// TIA Portal V20 export
DATA_BLOCK "DB_OPC_Laser"   // DB125
{ S7_Optimized_Access := 'TRUE' }
// stored: MemoryReserve 100
   VAR
      Scanner : Struct
         In : Struct
            CheckNumber : Byte;
            Ready : Bool;
            Status : DInt;
            StatusDescription : String;
         END_STRUCT;
         Out : Struct
            Parameters : Struct
               IsFirstJobOfPiece : Bool;
               StationNumber : Byte;
               HoleNumber : DInt;
               JobListName : String;
               JobName : String;
               MeasureZ : LReal;
            END_STRUCT;
            RequestJob : Bool;
            CheckNumber : Byte;
         END_STRUCT;
      END_STRUCT;
   END_VAR
BEGIN
END_DATA_BLOCK
